ABB RAPID module: Module1.mod

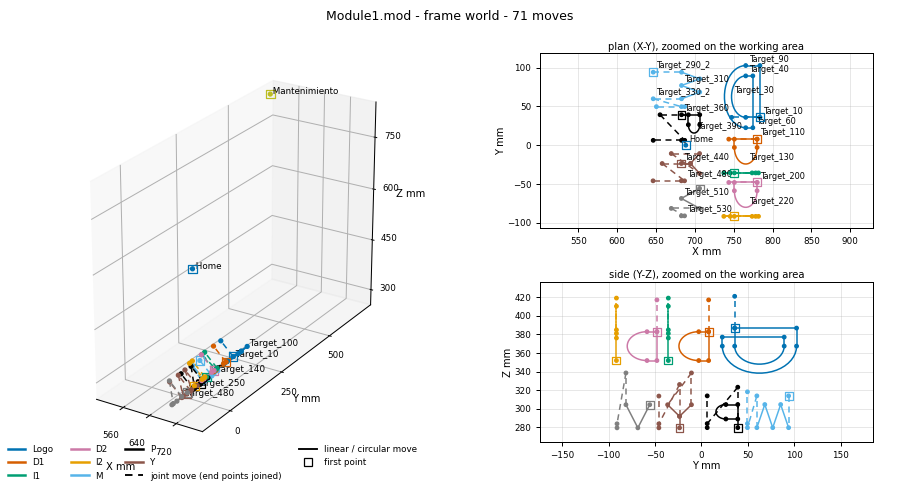
[picture p0: tool path of Module1.mod in frame world, 71 of 71 moves have a stored position in this frame; points joined in program order, loops and branches not executed]
MODULE Module1
    CONST robtarget Target_360:=[[193.374,164.249,0],[1,0,0,0],[0,-2,1,0],[9E+09,9E+09,9E+09,9E+09,9E+09,9E+09]];
    CONST robtarget Target_370:=[[159.174,164.249,0],[1,0,0,0],[0,-2,1,0],[9E+09,9E+09,9E+09,9E+09,9E+09,9E+09]];
    CONST robtarget Target_380:=[[159.174,151.424,0],[1,0,0,0],[0,-2,1,0],[9E+09,9E+09,9E+09,9E+09,9E+09,9E+09]];
    CONST robtarget Target_410:=[[180.549,164.249,0],[1,0,0,0],[0,-2,1,0],[9E+09,9E+09,9E+09,9E+09,9E+09,9E+09]];
    CONST robtarget Target_390:=[[169.861,140.736,0],[1,0,0,0],[0,-2,1,0],[9E+09,9E+09,9E+09,9E+09,9E+09,9E+09]];
    CONST robtarget Target_400:=[[180.549,151.424,0],[1,0,0,0],[0,-2,1,0],[9E+09,9E+09,9E+09,9E+09,9E+09,9E+09]];
    CONST robtarget Target_420:=[[187.389,131.33,0],[1,0,0,0],[0,-2,1,0],[9E+09,9E+09,9E+09,9E+09,9E+09,9E+09]];
    CONST robtarget Target_430:=[[193.374,131.33,0],[1,0,0,0],[0,-2,1,0],[9E+09,9E+09,9E+09,9E+09,9E+09,9E+09]];
    CONST robtarget Target_440:=[[193.651,101.513,0],[1,0,0,0],[-1,1,-2,0],[9E+09,9E+09,9E+09,9E+09,9E+09,9E+09]];
    CONST robtarget Target_450:=[[176.551,101.513,0],[1,0,0,0],[-1,1,-2,0],[9E+09,9E+09,9E+09,9E+09,9E+09,9E+09]];
    CONST robtarget Target_550:=[[171.613,66,0],[1,0,0,0],[0,-2,1,0],[9E+09,9E+09,9E+09,9E+09,9E+09,9E+09]];
    CONST robtarget Target_560:=[[171.613,81,0],[1,0,0,0],[0,-2,1,0],[9E+09,9E+09,9E+09,9E+09,9E+09,9E+09]];
    CONST robtarget Target_570:=[[179.613,46.5,0],[1,0,0,0],[0,-2,1,0],[9E+09,9E+09,9E+09,9E+09,9E+09,9E+09]];
    CONST robtarget Target_580:=[[186.613,46.5,0],[1,0,0,0],[0,-2,1,0],[9E+09,9E+09,9E+09,9E+09,9E+09,9E+09]];
    CONST robtarget Target_590:=[[214.649,187,0],[1,0,0,0],[0,0,0,0],[9E+09,9E+09,9E+09,9E+09,9E+09,9E+09]];
    CONST robtarget Target_620:=[[254.649,172,0],[1,0,0,0],[0,-2,1,0],[9E+09,9E+09,9E+09,9E+09,9E+09,9E+09]];
    CONST robtarget Target_600:=[[234.649,172,0],[1,0,0,0],[0,-2,1,0],[9E+09,9E+09,9E+09,9E+09,9E+09,9E+09]];
    CONST robtarget Target_610:=[[214.649,157,0],[1,0,0,0],[0,-2,1,0],[9E+09,9E+09,9E+09,9E+09,9E+09,9E+09]];
    CONST robtarget Target_630:=[[247.649,150,0],[1,0,0,0],[0,0,0,0],[9E+09,9E+09,9E+09,9E+09,9E+09,9E+09]];
    CONST robtarget Target_10:=[[46.091,160.915,0],[1,0,0,0],[0,-1,0,0],[9E+09,9E+09,9E+09,9E+09,9E+09,9E+09]];
    CONST robtarget Target_20:=[[72.767,160.915,0],[1,0,0,0],[0,0,0,0],[9E+09,9E+09,9E+09,9E+09,9E+09,9E+09]];
    CONST robtarget Target_30:=[[99.443,187.591,0],[1,0,0,0],[0,-1,0,0],[9E+09,9E+09,9E+09,9E+09,9E+09,9E+09]];
    CONST robtarget Target_40:=[[72.767,214.267,0],[1,0,0,0],[0,-1,0,0],[9E+09,9E+09,9E+09,9E+09,9E+09,9E+09]];
    CONST robtarget Target_50:=[[59.429,214.267,0],[1,0,0,0],[0,-1,0,0],[9E+09,9E+09,9E+09,9E+09,9E+09,9E+09]];
    CONST robtarget Target_60:=[[59.429,147.577,0],[1,0,0,0],[0,-1,0,0],[9E+09,9E+09,9E+09,9E+09,9E+09,9E+09]];
    CONST robtarget Target_70:=[[72.767,147.577,0],[1,0,0,0],[0,-1,0,0],[9E+09,9E+09,9E+09,9E+09,9E+09,9E+09]];
    CONST robtarget Target_80:=[[112.781,187.591,0],[1,0,0,0],[0,-1,0,0],[9E+09,9E+09,9E+09,9E+09,9E+09,9E+09]];
    CONST robtarget Target_90:=[[72.767,227.605,0],[1,0,0,0],[0,-1,0,0],[9E+09,9E+09,9E+09,9E+09,9E+09,9E+09]];
    CONST robtarget Target_100:=[[46.091,227.605,0],[1,0,0,0],[0,-1,0,0],[9E+09,9E+09,9E+09,9E+09,9E+09,9E+09]];
    CONST robtarget Target_310:=[[193.374,201.918,0],[1,0,0,0],[0,-2,1,0],[9E+09,9E+09,9E+09,9E+09,9E+09,9E+09]];
    CONST robtarget Target_110:=[[51.426,132.866,0],[1,0,0,0],[0,0,0,0],[9E+09,9E+09,9E+09,9E+09,9E+09,9E+09]];
    CONST robtarget Target_120:=[[51.426,122.195,0],[1,0,0,0],[-1,0,-1,0],[9E+09,9E+09,9E+09,9E+09,9E+09,9E+09]];
    CONST robtarget Target_130:=[[72.767,100.855,0],[1,0,0,0],[-1,0,-1,0],[9E+09,9E+09,9E+09,9E+09,9E+09,9E+09]];
    CONST robtarget Target_140:=[[94.108,122.195,0],[1,0,0,0],[-1,0,-1,0],[9E+09,9E+09,9E+09,9E+09,9E+09,9E+09]];
    CONST robtarget Target_150:=[[94.108,132.866,0],[1,0,0,0],[0,-1,0,0],[9E+09,9E+09,9E+09,9E+09,9E+09,9E+09]];
    CONST robtarget Target_320:=[[159.174,193.368,0],[1,0,0,0],[0,-1,1,0],[9E+09,9E+09,9E+09,9E+09,9E+09,9E+09]];
    CONST robtarget Target_160:=[[94.108,89.421,0],[1,0,0,0],[0,0,0,0],[9E+09,9E+09,9E+09,9E+09,9E+09,9E+09]];
    CONST robtarget Target_170:=[[60.763,89.421,0],[1,0,0,0],[-1,0,-1,0],[9E+09,9E+09,9E+09,9E+09,9E+09,9E+09]];
    CONST robtarget Target_200:=[[51.426,77.138,0],[1,0,0,0],[0,0,0,0],[9E+09,9E+09,9E+09,9E+09,9E+09,9E+09]];
    CONST robtarget Target_180:=[[54.094,89.421,0],[1,0,0,0],[-1,0,-1,0],[9E+09,9E+09,9E+09,9E+09,9E+09,9E+09]];
    CONST robtarget Target_190:=[[48.759,89.421,0],[1,0,0,0],[-1,0,-1,0],[9E+09,9E+09,9E+09,9E+09,9E+09,9E+09]];
    CONST robtarget Target_330:=[[193.374,184.818,0],[1,0,0,0],[0,-2,1,0],[9E+09,9E+09,9E+09,9E+09,9E+09,9E+09]];
    CONST robtarget Target_220:=[[72.767,45.127,0],[1,0,0,0],[-1,0,-1,0],[9E+09,9E+09,9E+09,9E+09,9E+09,9E+09]];
    CONST robtarget Target_230:=[[94.108,66.467,0],[1,0,0,0],[-1,0,-1,0],[9E+09,9E+09,9E+09,9E+09,9E+09,9E+09]];
    CONST robtarget Target_240:=[[94.108,77.138,0],[1,0,0,0],[-1,0,-1,0],[9E+09,9E+09,9E+09,9E+09,9E+09,9E+09]];
    CONST robtarget Target_250:=[[94.108,33.511,0],[1,0,0,0],[0,0,0,0],[9E+09,9E+09,9E+09,9E+09,9E+09,9E+09]];
    CONST robtarget Target_210:=[[51.426,66.467,0],[1,0,0,0],[-1,0,-1,0],[9E+09,9E+09,9E+09,9E+09,9E+09,9E+09]];
    CONST robtarget Target_340:=[[193.374,174.678,0],[1,0,0,0],[0,-2,1,0],[9E+09,9E+09,9E+09,9E+09,9E+09,9E+09]];
    CONST robtarget Target_290:=[[193.374,219.018,0],[1,0,0,0],[0,0,0,0],[9E+09,9E+09,9E+09,9E+09,9E+09,9E+09]];
    CONST robtarget Target_280:=[[48.759,33.511,0],[1,0,0,0],[-1,0,-1,0],[9E+09,9E+09,9E+09,9E+09,9E+09,9E+09]];
    CONST robtarget Target_300:=[[159.174,210.468,0],[1,0,0,0],[0,-1,1,0],[9E+09,9E+09,9E+09,9E+09,9E+09,9E+09]];
    CONST robtarget Target_270:=[[54.094,33.511,0],[1,0,0,0],[-1,0,-1,0],[9E+09,9E+09,9E+09,9E+09,9E+09,9E+09]];
    CONST robtarget Target_260:=[[60.763,33.511,0],[1,0,0,0],[-1,0,-1,0],[9E+09,9E+09,9E+09,9E+09,9E+09,9E+09]];
    CONST robtarget Target_350:=[[187.389,174.678,0],[1,0,0,0],[0,-2,1,0],[9E+09,9E+09,9E+09,9E+09,9E+09,9E+09]];
    CONST robtarget Target_460:=[[159.451,114.338,0],[1,0,0,0],[-1,1,-2,0],[9E+09,9E+09,9E+09,9E+09,9E+09,9E+09]];
    CONST robtarget Target_470:=[[159.451,88.688,0],[1,0,0,0],[-1,1,-2,0],[9E+09,9E+09,9E+09,9E+09,9E+09,9E+09]];
    CONST robtarget Target_480:=[[187.666,79.24,0],[1,0,0,0],[-1,1,-2,0],[9E+09,9E+09,9E+09,9E+09,9E+09,9E+09]];
    CONST robtarget Target_490:=[[193.651,79.24,0],[1,0,0,0],[-1,1,-2,0],[9E+09,9E+09,9E+09,9E+09,9E+09,9E+09]];
    CONST robtarget Target_500:=[[159.451,69.411,0],[1,0,0,0],[-1,1,-2,0],[9E+09,9E+09,9E+09,9E+09,9E+09,9E+09]];
    CONST robtarget Target_530:=[[187.666,34.148,0],[1,0,0,0],[-1,1,-2,0],[9E+09,9E+09,9E+09,9E+09,9E+09,9E+09]];
    CONST robtarget Target_510:=[[193.651,56.586,0],[1,0,0,0],[-1,1,-2,0],[9E+09,9E+09,9E+09,9E+09,9E+09,9E+09]];
    CONST robtarget Target_520:=[[159.451,43.761,0],[1,0,0,0],[-1,0,-2,0],[9E+09,9E+09,9E+09,9E+09,9E+09,9E+09]];
    CONST robtarget Target_540:=[[193.651,34.148,0],[1,0,0,0],[-1,1,-2,0],[9E+09,9E+09,9E+09,9E+09,9E+09,9E+09]];
    CONST robtarget Target_640:=[[254.649,150,0],[1,0,0,0],[0,0,0,0],[9E+09,9E+09,9E+09,9E+09,9E+09,9E+09]];
    CONST robtarget Target_650:=[[214.649,143,0],[1,0,0,0],[-1,0,-1,0],[9E+09,9E+09,9E+09,9E+09,9E+09,9E+09]];
    CONST robtarget Target_660:=[[254.649,128,0],[1,0,0,0],[-1,0,-1,0],[9E+09,9E+09,9E+09,9E+09,9E+09,9E+09]];
    CONST robtarget Target_670:=[[214.649,113,0],[1,0,0,0],[-1,0,-1,0],[9E+09,9E+09,9E+09,9E+09,9E+09,9E+09]];
    CONST robtarget Target_680:=[[247.649,106,0],[1,0,0,0],[-1,0,-1,0],[9E+09,9E+09,9E+09,9E+09,9E+09,9E+09]];
    CONST robtarget Target_690:=[[254.649,106,0],[1,0,0,0],[-1,0,-1,0],[9E+09,9E+09,9E+09,9E+09,9E+09,9E+09]];
    CONST robtarget Target_720:=[[171.614154806,58.991203706,-36.638059024],[1,-0.000000034,0.000000051,-0.000000007],[0,-2,1,0],[9E+09,9E+09,9E+09,9E+09,9E+09,9E+09]];
    CONST robtarget Target_700:=[[179.614,46.5,0],[1,0,0,0],[0,-2,1,0],[9E+09,9E+09,9E+09,9E+09,9E+09,9E+09]];
    CONST robtarget Target_710:=[[186.614,46.5,0],[1,0,0,0],[0,-2,1,0],[9E+09,9E+09,9E+09,9E+09,9E+09,9E+09]];
    CONST robtarget Target_730:=[[206.575839686,130.575385522,-36.062606272],[1,-0.000000061,0.000000016,-0.000000213],[0,-2,1,0],[9E+09,9E+09,9E+09,9E+09,9E+09,9E+09]];
    CONST robtarget Target_740:=[[214.649,187,0],[1,0,0,0],[0,0,0,0],[9E+09,9E+09,9E+09,9E+09,9E+09,9E+09]];
    CONST robtarget Target_750:=[[234.649,172,0],[1,0,0,0],[0,-2,1,0],[9E+09,9E+09,9E+09,9E+09,9E+09,9E+09]];
    CONST robtarget Target_760:=[[214.649,157,0],[1,0,0,0],[0,-2,1,0],[9E+09,9E+09,9E+09,9E+09,9E+09,9E+09]];
    CONST robtarget Target_800:=[[224.454054793,169.052592344,-39.983761207],[1,-0.000000024,0.000000053,-0.000000097],[0,-2,1,0],[9E+09,9E+09,9E+09,9E+09,9E+09,9E+09]];
    CONST robtarget Target_770:=[[254.649,172,0],[1,0,0,0],[0,-2,1,0],[9E+09,9E+09,9E+09,9E+09,9E+09,9E+09]];
    CONST robtarget Target_810:=[[254.649337072,159.007769138,-30.298077251],[1,-0.000000027,0.000000051,-0.000000098],[0,-2,1,0],[9E+09,9E+09,9E+09,9E+09,9E+09,9E+09]];
    CONST robtarget Target_790:=[[254.649,150,0],[1,0,0,0],[0,-2,1,0],[9E+09,9E+09,9E+09,9E+09,9E+09,9E+09]];
    CONST robtarget Target_780:=[[247.649,150,0],[1,0,0,0],[0,-2,1,0],[9E+09,9E+09,9E+09,9E+09,9E+09,9E+09]];
    CONST robtarget Target_820:=[[229.743211704,145.004792269,-27.634877565],[1,-0.000000014,0.000000023,0.000000082],[0,-2,1,0],[9E+09,9E+09,9E+09,9E+09,9E+09,9E+09]];
    CONST robtarget Target_830:=[[214.649,143,0],[1,0,0,0],[0,0,0,0],[9E+09,9E+09,9E+09,9E+09,9E+09,9E+09]];
    CONST robtarget Target_840:=[[254.649,128,0],[1,0,0,0],[0,-2,1,0],[9E+09,9E+09,9E+09,9E+09,9E+09,9E+09]];
    CONST robtarget Target_850:=[[214.649,113,0],[1,0,0,0],[0,-2,1,0],[9E+09,9E+09,9E+09,9E+09,9E+09,9E+09]];
    CONST robtarget Target_880:=[[232.237809143,110.203682172,-19.826551886],[1,-0.000000178,0.000000032,0.000000095],[0,-2,1,0],[9E+09,9E+09,9E+09,9E+09,9E+09,9E+09]];
    CONST robtarget Target_860:=[[247.649,106,0],[1,0,0,0],[0,-2,1,0],[9E+09,9E+09,9E+09,9E+09,9E+09,9E+09]];
    CONST robtarget Target_870:=[[254.649,106,0],[1,0,0,0],[0,-2,1,0],[9E+09,9E+09,9E+09,9E+09,9E+09,9E+09]];
    CONST robtarget Home:=[[688.354427157,0,618.841978046],[0.5,0,0.866025404,0],[0,0,0,0],[9E+09,9E+09,9E+09,9E+09,9E+09,9E+09]];
    TASK PERS wobjdata Workobject_1:=[FALSE,TRUE,"",[[822.628,-125,413.586],[0.396843374,0,0.917886342,0]],[[0,0,-10],[1,0,0,0]]];
    CONST robtarget Target_900:=[[614.368006487,-305.026841829,-535.49276156],[0.482962895,-0.129409515,-0.299950184,0.812422247],[-1,0,0,0],[9E+09,9E+09,9E+09,9E+09,9E+09,9E+09]];
    CONST robtarget Target_910:=[[186.613,263,0],[1,0,0,0],[0,0,0,0],[9E+09,9E+09,9E+09,9E+09,9E+09,9E+09]];
    CONST robtarget Target_920:=[[146.613,248,0],[1,0,0,0],[0,0,-1,0],[9E+09,9E+09,9E+09,9E+09,9E+09,9E+09]];
    CONST robtarget Target_930:=[[186.613,233,0],[1,0,0,0],[0,0,-1,0],[9E+09,9E+09,9E+09,9E+09,9E+09,9E+09]];
    CONST robtarget Target_930_4:=[[186.613,233,-25],[1,0,0,0],[0,0,-1,0],[9E+09,9E+09,9E+09,9E+09,9E+09,9E+09]];
    CONST robtarget Target_940:=[[166.613,255.5,0],[1,0,0,0],[0,0,-1,0],[9E+09,9E+09,9E+09,9E+09,9E+09,9E+09]];
    CONST robtarget Target_950:=[[166.613,240.5,0],[1,0,0,0],[0,0,-1,0],[9E+09,9E+09,9E+09,9E+09,9E+09,9E+09]];
    CONST robtarget Target_950_2:=[[166.613,240.5,-25],[1,0,0,0],[0,0,-1,0],[9E+09,9E+09,9E+09,9E+09,9E+09,9E+09]];
    CONST robtarget Target_970:=[[179.613,226,0],[1,0,0,0],[0,0,-1,0],[9E+09,9E+09,9E+09,9E+09,9E+09,9E+09]];
    CONST robtarget Target_960:=[[186.613,226,0],[1,0,0,0],[0,0,-1,0],[9E+09,9E+09,9E+09,9E+09,9E+09,9E+09]];
    CONST robtarget Target_960_2:=[[186.613,226,-25],[1,0,0,0],[0,0,-1,0],[9E+09,9E+09,9E+09,9E+09,9E+09,9E+09]];
    CONST robtarget Target_mantenimiento:=[[-146.986419067,502.304411342,-380.503407182],[0.711946398,-0.412986595,-0.552472154,-0.131715289],[0,-1,0,1],[9E+09,9E+09,9E+09,9E+09,9E+09,9E+09]];
    PERS tooldata FinalTool:=[TRUE,[[-38.5,0,181],[1,0,0,0]],[1,[0,0,1],[1,0,0,0],0,0,0]];
    CONST robtarget Target_20_2:=[[43.067,178.883,-30],[1,0,0,0],[0,-1,0,0],[9E+09,9E+09,9E+09,9E+09,9E+09,9E+09]];
    CONST robtarget Target_120_2:=[[49.307,146.077,-30],[1,0,0,0],[0,-1,0,0],[9E+09,9E+09,9E+09,9E+09,9E+09,9E+09]];
    CONST robtarget Target_180_2:=[[52.427,99.277,-30],[1,0,0,0],[0,-1,0,0],[9E+09,9E+09,9E+09,9E+09,9E+09,9E+09]];
    CONST robtarget Target_200_2:=[[51.426,77.138,-50],[1,0,0,0],[-1,0,-1,0],[9E+09,9E+09,9E+09,9E+09,9E+09,9E+09]];
    CONST robtarget Target_220_2:=[[99.227,89.917,-30],[1,0,0,0],[0,-1,1,0],[9E+09,9E+09,9E+09,9E+09,9E+09,9E+09]];
    CONST robtarget Target_280_2:=[[48.759,33.511,-50],[1,0,0,0],[-1,0,-1,0],[9E+09,9E+09,9E+09,9E+09,9E+09,9E+09]];
    CONST robtarget Target_450_2:=[[176.551,101.513,-50],[1,0,0,0],[-1,0,-1,0],[9E+09,9E+09,9E+09,9E+09,9E+09,9E+09]];
    CONST robtarget Target_320_2:=[[186.613,233,-30],[1,0,0,0],[0,-1,1,0],[9E+09,9E+09,9E+09,9E+09,9E+09,9E+09]];
    CONST robtarget Target_340_2:=[[166.613,240.5,-30],[1,0,0,0],[0,-1,1,0],[9E+09,9E+09,9E+09,9E+09,9E+09,9E+09]];
    CONST robtarget Target_350_2:=[[187.389,174.678,-50],[1,0,0,0],[0,-1,0,0],[9E+09,9E+09,9E+09,9E+09,9E+09,9E+09]];
    CONST robtarget Target_410_2:=[[180.549,164.249,-50],[1,0,0,0],[0,-1,0,0],[9E+09,9E+09,9E+09,9E+09,9E+09,9E+09]];
    CONST robtarget Target_430_2:=[[193.374,131.33,-50],[1,0,0,0],[0,-1,0,0],[9E+09,9E+09,9E+09,9E+09,9E+09,9E+09]];
    CONST robtarget Target_480_2:=[[186.613,95,-30],[1,0,0,0],[0,-2,1,0],[9E+09,9E+09,9E+09,9E+09,9E+09,9E+09]];
    CONST robtarget Target_490_2:=[[193.651,79.24,-50],[1,0,0,0],[-1,0,-1,0],[9E+09,9E+09,9E+09,9E+09,9E+09,9E+09]];
    CONST robtarget Target_560_2:=[[171.613,81,-30],[1,0,0,0],[0,-2,1,0],[9E+09,9E+09,9E+09,9E+09,9E+09,9E+09]];
    CONST robtarget Target_580_2:=[[186.613,46.5,-30],[1,0,0,0],[0,-2,1,0],[9E+09,9E+09,9E+09,9E+09,9E+09,9E+09]];
    CONST robtarget Target_610_2:=[[214.649,157,-30],[1,0,0,0],[0,-2,1,0],[9E+09,9E+09,9E+09,9E+09,9E+09,9E+09]];
    CONST robtarget Target_620_2:=[[254.649,172,-30],[1,0,0,0],[0,-2,1,0],[9E+09,9E+09,9E+09,9E+09,9E+09,9E+09]];
    CONST robtarget Target_630_2:=[[247.649,150,-30],[1,0,0,0],[0,0,0,0],[9E+09,9E+09,9E+09,9E+09,9E+09,9E+09]];
    CONST robtarget Target_670_2:=[[214.649,113,-30],[1,0,0,0],[-1,0,-1,0],[9E+09,9E+09,9E+09,9E+09,9E+09,9E+09]];
    CONST robtarget Mantenimiento:=[[491.434141762,691.445179965,824.691178836],[0.866840807,-0.149108085,0.220825114,0.42141436],[0,-1,0,1],[9E+09,9E+09,9E+09,9E+09,9E+09,9E+09]];
    CONST robtarget Target_10_2:=[[46.091,160.915,-50],[1,0,0,0],[0,-1,0,0],[9E+09,9E+09,9E+09,9E+09,9E+09,9E+09]];
    CONST robtarget Target_110_2:=[[51.426,132.866,-50],[1,0,0,0],[0,-1,0,0],[9E+09,9E+09,9E+09,9E+09,9E+09,9E+09]];
    CONST robtarget Target_170_2:=[[60.763,89.421,-50],[1,0,0,0],[-1,0,-1,0],[9E+09,9E+09,9E+09,9E+09,9E+09,9E+09]];
    CONST robtarget Target_190_2:=[[48.759,89.421,-50],[1,0,0,0],[-1,0,-1,0],[9E+09,9E+09,9E+09,9E+09,9E+09,9E+09]];
    CONST robtarget Target_260_2:=[[60.763,33.511,-50],[1,0,0,0],[-1,0,-1,0],[9E+09,9E+09,9E+09,9E+09,9E+09,9E+09]];
    CONST robtarget Target_290_2:=[[193.374,219.018,-50],[1,0,0,0],[0,-1,1,0],[9E+09,9E+09,9E+09,9E+09,9E+09,9E+09]];
    CONST robtarget Target_330_2:=[[193.374,184.818,-50],[1,0,0,0],[0,-1,0,0],[9E+09,9E+09,9E+09,9E+09,9E+09,9E+09]];
    CONST robtarget Target_460_2:=[[159.451,114.338,-50],[1,0,0,0],[-1,0,-1,0],[9E+09,9E+09,9E+09,9E+09,9E+09,9E+09]];
    CONST robtarget Target_520_2:=[[159.451,43.761,-50],[1,0,0,0],[-1,0,-1,0],[9E+09,9E+09,9E+09,9E+09,9E+09,9E+09]];

    PROC Logo()
        MoveJ Target_10,v100,fine,FinalTool\WObj:=Workobject_1;
        MoveL Target_20,v100,fine,FinalTool\WObj:=Workobject_1;
        MoveC Target_30,Target_40,v100,fine,FinalTool\WObj:=Workobject_1;
        MoveL Target_50,v100,fine,FinalTool\WObj:=Workobject_1;
        MoveL Target_60,v100,fine,FinalTool\WObj:=Workobject_1;
        MoveL Target_70,v100,fine,FinalTool\WObj:=Workobject_1;
        MoveC Target_80,Target_90,v100,fine,FinalTool\WObj:=Workobject_1;
        MoveL Target_100,v100,fine,FinalTool\WObj:=Workobject_1;
        MoveL Target_10,v100,fine,FinalTool\WObj:=Workobject_1;
        MoveJ Target_10_2,v200,z10,FinalTool\WObj:=Workobject_1;

    ENDPROC
    PROC D1()
        MoveJ Target_110,v100,fine,FinalTool\WObj:=Workobject_1;
        MoveL Target_120,v100,fine,FinalTool\WObj:=Workobject_1;
        MoveC Target_130,Target_140,v100,fine,FinalTool\WObj:=Workobject_1;
        MoveL Target_150,v100,fine,FinalTool\WObj:=Workobject_1;
        MoveL Target_110,v100,fine,FinalTool\WObj:=Workobject_1;
        MoveJ Target_110_2,v200,z10,FinalTool\WObj:=Workobject_1;

    ENDPROC
    PROC I1()
        MoveJ Target_160,v100,fine,FinalTool\WObj:=Workobject_1;
        MoveL Target_170,v100,fine,FinalTool\WObj:=Workobject_1;
        MoveJ Target_170_2,v200,z10,FinalTool\WObj:=Workobject_1;
        MoveJ Target_180,v100,fine,FinalTool\WObj:=Workobject_1;
        MoveL Target_190,v100,fine,FinalTool\WObj:=Workobject_1;
        MoveJ Target_190_2,v200,z10,FinalTool\WObj:=Workobject_1;

    ENDPROC
    PROC D2()
        MoveJ Target_200,v100,fine,FinalTool\WObj:=Workobject_1;
        MoveL Target_210,v100,fine,FinalTool\WObj:=Workobject_1;
        MoveC Target_220,Target_230,v100,fine,FinalTool\WObj:=Workobject_1;
        MoveL Target_240,v100,fine,FinalTool\WObj:=Workobject_1;
        MoveL Target_200,v100,fine,FinalTool\WObj:=Workobject_1;
        MoveJ Target_200_2,v200,z10,FinalTool\WObj:=Workobject_1;

    ENDPROC
    PROC I2()
        MoveJ Target_250,v100,fine,FinalTool\WObj:=Workobject_1;
        MoveL Target_260,v100,fine,FinalTool\WObj:=Workobject_1;
        MoveJ Target_260_2,v200,z10,FinalTool\WObj:=Workobject_1;
        MoveJ Target_270,v100,fine,FinalTool\WObj:=Workobject_1;
        MoveL Target_280,v100,fine,FinalTool\WObj:=Workobject_1;
        MoveJ Target_280_2,v200,z10,FinalTool\WObj:=Workobject_1;
    ENDPROC

    PROC M()
        MoveJ Target_290_2,v200,z10,FinalTool\WObj:=Workobject_1;
        MoveJ Target_290,v100,fine,FinalTool\WObj:=Workobject_1;
        MoveL Target_300,v100,fine,FinalTool\WObj:=Workobject_1;
        MoveL Target_310,v100,fine,FinalTool\WObj:=Workobject_1;
        MoveL Target_320,v100,fine,FinalTool\WObj:=Workobject_1;
        MoveL Target_330,v100,fine,FinalTool\WObj:=Workobject_1;
        MoveJ Target_330_2,v200,z10,FinalTool\WObj:=Workobject_1;
        MoveJ Target_340,v100,fine,FinalTool\WObj:=Workobject_1;
        MoveL Target_350,v100,fine,FinalTool\WObj:=Workobject_1;
        MoveJ Target_350_2,v200,z10,FinalTool\WObj:=Workobject_1;
    ENDPROC

    PROC P()
        MoveJ Target_360,v100,fine,FinalTool\WObj:=Workobject_1;
        MoveL Target_370,v100,fine,FinalTool\WObj:=Workobject_1;
        MoveL Target_380,v100,fine,FinalTool\WObj:=Workobject_1;
        MoveC Target_390,Target_400,v100,fine,FinalTool\WObj:=Workobject_1;
        MoveL Target_410,v100,fine,FinalTool\WObj:=Workobject_1;
        MoveJ Target_410_2,v200,z10,FinalTool\WObj:=Workobject_1;
        MoveJ Target_420,v100,fine,FinalTool\WObj:=Workobject_1;
        MoveJ Target_430,v100,fine,FinalTool\WObj:=Workobject_1;
        MoveJ Target_430_2,v200,z10,FinalTool\WObj:=Workobject_1;

    ENDPROC
    PROC Y()
        MoveJ Target_440,v100,fine,FinalTool\WObj:=Workobject_1;
        MoveL Target_450,v100,fine,FinalTool\WObj:=Workobject_1;
        MoveL Target_460,v100,fine,FinalTool\WObj:=Workobject_1;
        MoveJ Target_460_2,v200,z10,FinalTool\WObj:=Workobject_1;
        MoveJ Target_470,v100,fine,FinalTool\WObj:=Workobject_1;
        MoveL Target_450,v100,fine,FinalTool\WObj:=Workobject_1;
        MoveJ Target_450_2,v200,z10,FinalTool\WObj:=Workobject_1;
        MoveJ Target_480,v100,fine,FinalTool\WObj:=Workobject_1;
        MoveL Target_490,v100,fine,FinalTool\WObj:=Workobject_1;
        MoveJ Target_490_2,v200,z10,FinalTool\WObj:=Workobject_1;

    ENDPROC
    PROC V()
        MoveJ Target_500,v100,fine,FinalTool\WObj:=Workobject_1;
        MoveL Target_510,v100,fine,FinalTool\WObj:=Workobject_1;
        MoveL Target_520,v100,fine,FinalTool\WObj:=Workobject_1;
        MoveJ Target_520_2,v200,z10,FinalTool\WObj:=Workobject_1;
        MoveJ Target_530,v100,fine,FinalTool\WObj:=Workobject_1;
        MoveL Target_540,v100,fine,FinalTool\WObj:=Workobject_1;

    ENDPROC

    PROC GoMantenimeinto()
        Homing;
        SetDO DO_03,0;
        SetDO DO_02,1;
        MoveJ Mantenimiento,v200,z10,FinalTool\WObj:=wobj0;
    ENDPROC

    PROC GoEscritura()
        Homing;
        SetDO DO_03,0;
        SetDO DO_01,1;
        Logo;
        D1;
        I1;
        D2;
        I2;
        M;
        P;
        Y;
        V;
    ENDPROC

    PROC Homing()
        SetDO DO_01,0;
        SetDO DO_02,0;
        SetDO DO_03,1;
        MoveJ Home,v300,z10,FinalTool\WObj:=wobj0;
    ENDPROC

    PROC Main()
        WHILE TRUE DO
            IF DI_01 = 1 THEN
                GoEscritura;
            ELSEIF DI_02 = 1 THEN
                GoMantenimeinto;
            ELSEIF DI_03 = 1 THEN
                Homing;
            ENDIF
        ENDWHILE
    ENDPROC
ENDMODULE
